Yaskawa INFORM job: R2_W39(-180_180).JBI

/JOB
//NAME R2_W39(-180_180)
///FOLDERNAME KR_OK
//POS
///NPOS 14,14,0,2,0,0
///TOOL 0
///POSTYPE PULSE
///PULSE
C00000=186873,-12127,-67877,2915,95406,54913
C00001=186848,-12081,-67842,2924,95409,54906
C00002=172444,-8158,-30910,19742,90226,52779
C00003=172444,-8236,-30399,19740,89894,52726
C00004=172444,-8158,-30910,19742,90226,52779
C00005=173273,-10458,-32717,19595,89969,53024
C00006=173273,-10588,-31826,19590,89387,52931
C00007=173050,-9983,-31354,19629,89459,52867
C00008=173273,-10588,-31826,19590,89387,52931
C00009=173273,-10228,-34028,19608,90842,53166
C00010=170325,-13683,-34381,20095,90062,52012
C00011=176033,-3267,-26149,19097,89007,53825
C00012=176033,-2899,-28274,19110,90425,54047
C00013=186848,-12081,-67842,2924,95409,54906
BC00000=335208,209816,1075201
BC00001=335208,132950,1075201
BC00002=335208,132950,1075201
BC00003=335208,132950,1075201
BC00004=335208,132950,1075201
BC00005=335208,132950,1075201
BC00006=335208,132950,1075201
BC00007=335208,132950,1075201
BC00008=335208,132950,1075201
BC00009=335208,132950,1075201
BC00010=335208,132950,1075201
BC00011=335208,132950,1075201
BC00012=335208,132950,1075201
BC00013=335208,132950,1075201
///POSTYPE BASE
///RECTAN
///RCONF 0,0,0,0,1,0,0,0,0,0,0,0,0,0,0,0,0,0,0,0,0,0,0,0
P00006=2.006,1.622,-0.565,0.0000,0.0000,0.0000
P00021=0.073,2.058,-0.109,0.0000,0.0000,0.0000
//INST
///DATE 2023/11/07 14:10
///ATTR SC,RW
///GROUP1 RB1,BS1
NOP
SFTOF
MOVJ C00000 BC00000 VJ=10.00
MOVJ C00001 BC00001 VJ=10.00
MOVL C00002 BC00002 V=100.0
REFP 3 C00003 BC00003
CALL JOB:SEARCH-R1
SET P021 P006
SFTON P021
MOVL C00004 BC00004 V=60.0
MOVL C00005 BC00005 V=60.0
MOVL C00006 BC00006 V=60.0
REFP 3 C00007 BC00007
CALL JOB:SEARCH-R1
SET P021 P006
SFTON P021
MOVL C00008 BC00008 V=60.0
MOVL C00009 BC00009 V=60.0
MOVL C00010 BC00010 V=25.0 PL=0
MACRO1 MJ#(0) ARGF6
ARCON
MOVL C00011 BC00011 V=11.7
ARCOF
MOVL C00012 BC00012 V=25.0
MOVJ C00013 BC00013 VJ=10.00
END
